FUNCTION_BLOCK FB_serializer
VAR_INPUT
END_VAR
VAR_OUTPUT
END_VAR
VAR
  fbJson  : FB_JsonSaxWriter;
END_VAR

METHOD serialize : STRING(255)
VAR_INPUT
  datetime: STRING;
  device_name: STRING;
  diag_data_body: POINTER TO sdo_xplanar_aps_diag;
END_VAR
fbJson.StartObject();       // ‘{‘ の出力
fbJson.AddKey('datetime');
fbJson.AddString(datetime);
fbJson.AddKey('device_name');
fbJson.AddString(device_name);
fbJson.AddKey('temperature');		//キー temperature: の出力
fbJson.AddUdint(diag_data_body^.temperature_center); // 温度出力
fbJson.AddKey('fan_rpm');		//キー temperature: の出力
fbJson.AddUdint(diag_data_body^.fan_rpm); // FAN回転数出力
fbJson.EndObject();			// ‘}’ の出力
serialize := fbJson.GetDocument();	// 文字列へ出力
fbJson.ResetDocument();		// SAXバッファクリア
END_METHOD

END_FUNCTION_BLOCK

(* stored: Version 1.1.0.1, ProductVersion 3.1.4024.12
   POU FB_serializer: Id {3882d52d-38c6-4913-93dc-840aaa8feded}, SpecialFunc None
   Method serialize: Id {74ef5bf3-cc3a-45e7-9e61-1ecdc904127b} *)
